// TIA Portal V20 export
FUNCTION_BLOCK "Fx_FbdLogic"   // FB3, FBD
{ S7_Optimized_Access := 'TRUE' }
// stored: MemoryReserve 100, SetENOAutomatically false
   VAR_INPUT
      "a" : Bool;
      "b" : Bool;
      c : Bool;
      n : Int;
   END_VAR
   VAR_OUTPUT
      and_ : Bool;
      or_ : Bool;
      xor_ : Bool;
      mix : Bool;
      held : Bool;
      big : Bool;
      late : Bool;
      latch : Bool;
   END_VAR
   VAR
      delay : TON_TIME;
      sr : Bool;
   END_VAR
BEGIN

REGION Network 1
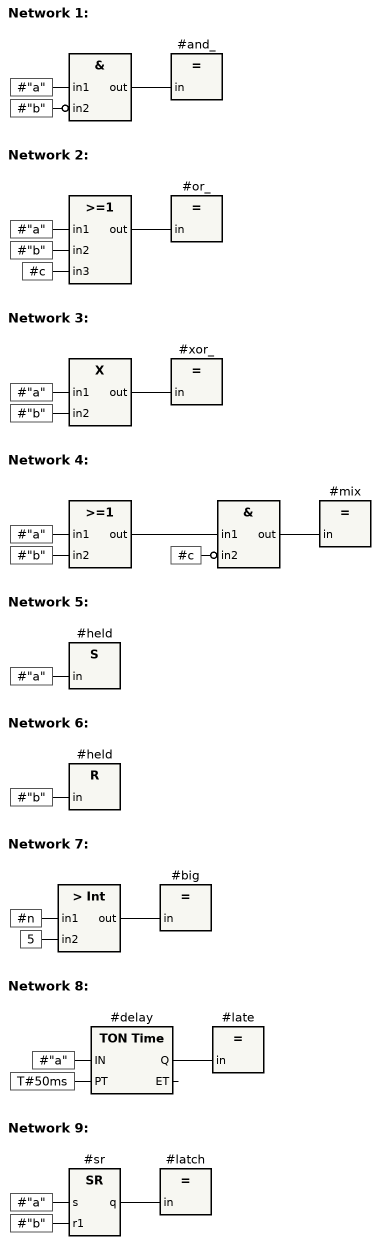
   #and_ := #"a" AND NOT #"b";
END_REGION

REGION Network 2
   #or_ := #"a" OR #"b" OR #c;
END_REGION

REGION Network 3
   #xor_ := #"a" XOR #"b";
END_REGION

REGION Network 4
   #mix := (#"a" OR #"b") AND NOT #c;
END_REGION

REGION Network 5
   IF #"a" THEN #held := TRUE; END_IF;
END_REGION

REGION Network 6
   IF #"b" THEN #held := FALSE; END_IF;
END_REGION

REGION Network 7
   #big := #n > 5;
END_REGION

REGION Network 8
   #delay(IN := #"a", PT := T#50ms);   // TON
   #late := #delay.Q;
END_REGION

REGION Network 9
   IF #"a" THEN
       #sr := TRUE;   // SR flip-flop
   END_IF;
   IF #"b" THEN #sr := FALSE; END_IF;
   #latch := #sr;
END_REGION
END_FUNCTION_BLOCK
